Staubli VAL3: userPage.pjx

--- userPage.pjx ---
Parameters version=s7.6.3 stackSize=5000 millimeterUnit=true
Program file=changeTrsf.pgx
Program file=changeValue.pgx
Program file=clear.pgx
Program file=divideString.pgx
Program file=editNumField.pgx
Program file=findPos.pgx
Program file=getListPosition.pgx
Program file=getMenu.pgx
Program file=getView.pgx
Program file=insertDialog.pgx
Program file=insertDialog1.pgx
Program file=isListEmpty.pgx
Program file=leftPos.pgx
Program file=listadd.pgx
Program file=listcreate.pgx
Program file=listcursor.pgx
Program file=listdel.pgx
Program file=listempty.pgx
Program file=listevent.pgx
Program file=listframe.pgx
Program file=listins.pgx
Program file=listredraw.pgx
Program file=listupdate.pgx
Program file=listupdate1.pgx
Program file=midPos.pgx
Program file=nullKey.pgx
Program file=numCopy.pgx
Program file=printScroll.pgx
Program file=questionDialog.pgx
Program file=read.pgx
Program file=rightPos.pgx
Program file=scroll.pgx
Program file=selectNewField.pgx
Program file=setCenter.pgx
Program file=setMenu.pgx
Program file=setSizeList.pgx
Program file=setView.pgx
Program file=showBoolStatus.pgx
Program file=strfill.pgx
Program file=strfillchr.pgx
Program file=stringCopy.pgx
Program file=stringToArray.pgx
Program file=stringToFxArray.pgx
Program file=strlength.pgx
Program file=timerDialog.pgx
Program file=type.pgx
Program file=typeCenter.pgx
Program file=typeLen.pgx
Program file=typeMenu.pgx
Program file=yes_no.pgx
Program file=yes_no_cancel.pgx
Data file=userPage.dtx

--- changeTrsf.pgx ---
public program changeTrsf(trsf& x_tTrsf[], string x_sTitle, string x_sComment)
  local string l_sEvent
  local num l_nIndex
  local num l_nView
  local bool l_bRefresh
  local string l_sMessage
  local trsf l_tTrsf
  local string l_sItem
  local string l_sEmpty
  local point l_pPoint
  local tool l_tTool
  local num l_nAddon
  local num l_nDistanceX
  local num l_nDistanceY
  local bool l_bCheck
  local joint l_jPoint
begin
  logMsg("[KERNEL] INTERFACE:PAGE changeTrsf "+x_sTitle)
  // INIT all
  l_bRefresh=false
  l_nIndex=0
  l_nView=0
  call setSizeList(19,0,19,8)
  call setView(false)
  l_tTrsf=x_tTrsf
  //release the button
  call nullKey(nKey)
  // set the frame
  do
    cls()
    call type(0,12,x_sComment)
    call typeMenu(8,"OK")
    call listcreate(x_sTitle)
    l_sItem=("coord  X > "+toString(".2",l_tTrsf.x))
    call listadd(l_sItem)
    l_sItem=("coord  Y > "+toString(".2",l_tTrsf.y))
    call listadd(l_sItem)
    l_sItem=("coord  Z > "+toString(".2",l_tTrsf.z))
    call listadd(l_sItem)
    l_sItem=("coord RX > "+toString(".2",l_tTrsf.rx))
    call listadd(l_sItem)
    l_sItem=("coord RY > "+toString(".2",l_tTrsf.ry))
    call listadd(l_sItem)
    l_sItem=("coord RZ > "+toString(".2",l_tTrsf.rz))
    call listadd(l_sItem)
    // show the list
    nView=l_nIndex
    call listupdate(l_nIndex-l_nView)
    do
      l_nView=nView
      nKey=get()
      l_pPoint.trsf=l_tTrsf
      call listevent(nKey,l_nIndex,l_sEvent)
      switch nKey
        case 270
          //
          // clean the line
          call listcursor(nView,false)
          l_sEmpty=""
          switch l_nIndex
            case 0
              //  x-value
              call changeValue(l_tTrsf.x,0,0,10+40-nBottomX,nView+1,l_sEmpty)
            break
            case 1
              //  y-value
              call changeValue(l_tTrsf.y,0,0,10+40-nBottomX,nView+1,l_sEmpty)
            break
            case 2
              //  z-value
              call changeValue(l_tTrsf.z,0,0,10+40-nBottomX,nView+1,l_sEmpty)
            break
            case 3
              //  rx-value
              call changeValue(l_tTrsf.rx,0,0,10+40-nBottomX,nView+1,l_sEmpty)
            break
            case 4
              //  ry-value
              call changeValue(l_tTrsf.ry,0,0,10+40-nBottomX,nView+1,l_sEmpty)
            break
            case 5
              //  rz-value
              call changeValue(l_tTrsf.rz,0,0,10+40-nBottomX,nView+1,l_sEmpty)
            break
            case 6
              // addon
              l_nIndex=find(l_sEvent,">")
              call changeValue(l_nAddon,0,0,l_nIndex+1+2+nTopX,nView+nTopY+1,l_sEmpty)
            break
          endSwitch
          l_bRefresh=true
        break
        case 278
          // VALIDATE
          x_tTrsf=l_tTrsf
        break
      endSwitch
    until l_bRefresh==true or nKey==255 or nKey==278
    l_bRefresh=false
  until nKey==255 or nKey==278
  // check the key
  if nKey==278
    // validate
    x_tTrsf=l_tTrsf
  endIf
  // release the resource
  call nullKey(nKey)
end

--- changeValue.pgx ---
public program changeValue(num& x_nValue[], num x_nMin, num x_nMax, num x_nX, num x_nY, string& x_sItems[])
  local num l_nOldValue[2]
  local string l_sItem
  local string l_sMessage
  local bool l_bComma
  local string l_sEmpty
begin
  //---------------------------------
  // Staubli copyright 2005
  //                By toneage
  //[Public]-------------------------
  //
  // x_nValue:  num to change
  // x_nMax:    max value
  // x_nMin:    min value
  // x_nX:      X position
  // x_nY:      Y position
  // x_sItems   message
  //
  // look if the value is between max and min
  //
  if x_nMin>x_nMax
    return
  endIf
  //
  // print the line in white
  //
  // call listCleanLine()
  //
  call nullKey(nKey)
  l_nOldValue[1]=round(x_nValue)
  x_nValue=(round(x_nValue*100))/100
  l_nOldValue=x_nValue
  // check if is using the comma or not
  if l_nOldValue!=l_nOldValue[1]
    l_bComma=true
  else
    l_bComma=false
  endIf
  // start
  call clear(0,13)
  do
    if x_sItems==""
      //
      //  use the get num
      //
      if l_bComma
        call strfill(l_sEmpty,len(toString(".2",x_nValue)),l_sEmpty)
      else
        call strfill(l_sEmpty,len(toString("",x_nValue)),l_sEmpty)
      endIf
      call type(x_nX,x_nY,l_sEmpty)
      gotoxy(x_nX,x_nY)
      nKey=get(x_nValue)
      // check the comma again
      if round(x_nValue)!=x_nValue
        l_bComma=true
      endIf
      //
      // CHECK for MIN MAX VALUE
      //
      if x_nMax!=x_nMin or x_nMin!=0
        if x_nValue>x_nMax
          //
          // ask if you want to continue
          //
          popUpMsg("MAX: "+toString(".2",x_nMax))
          x_nValue=l_nOldValue
          //x_nValue=x_nMax
          nKey=-1
        else
          if x_nValue<x_nMin
            //
            popUpMsg("MIN: "+toString(".2",x_nMin))
            //x_nValue=x_nMin
            x_nValue=l_nOldValue
            nKey=-1
          endIf
        endIf
      endIf
      //
      // UPDATE THE VALUE
      //
      if l_bComma
        call type(x_nX,x_nY,toString(".2",x_nValue))
      else
        call type(x_nX,x_nY,toString("",x_nValue))
      endIf
    else
      //
      // STRING CHOICE
      //
      // show a list if there is the place
      call setSizeList(x_nX-1,max(0,x_nY-1),40-x_nX-1,min(13-x_nY,size(x_sItems)))
      call listcreate("")
      call listadd(x_sItems)
      call selectNewField(x_nValue,x_nValue,0)
      do
        nKey=get()
        call listevent(nKey,x_nValue,l_sItem)
      until nKey==270 or nKey==255
    endIf
  until nKey==270 or nKey==255
  if nKey==255
    bUseEscape=true
    x_nValue=l_nOldValue
    if x_sItems!=""
      x_sItems=x_sItems[l_nOldValue]
    endIf
  else
    bUseEscape=false
  endIf
end

--- insertDialog1.pgx ---
public program insertDialog1(string x_sMsg, num& x_nItem[], num x_nMin, num x_nMax)
  local num l_nStartLine
  local num l_nLine
  local num i
  local num l_nPX
  local num l_nPY
  local string l_sItem
  local string l_sMessage
  local string l_sEmpty
begin
  //
  // modify the x_sItem, using a min max range
  //
  if watch(bShowDialog==false,3)==false
    bShowDialog=false
    return
  else
    setMutex(bShowDialog)
    // clear the line
    call clear(0,13)
    // look for the comma
    if round(x_nItem)!=x_nItem
      l_sItem=toString(".2",x_nItem)
    else
      l_sItem=toString("",x_nItem)
    endIf
    // print the line
    l_sItem=x_sMsg+">"+l_sItem
    call stringCopy(l_sItem,sMessage)
    // divide the sentence
    call divideString(sMessage,l_nLine)
    l_nStartLine=round(5-l_nLine/2)
    // Start LINE
    call type(0,l_nStartLine-2,"┌──────────────────────────────────────┐")
    call type(0,l_nStartLine-1,"│                                      │")
    // write the message
    for i=0 to l_nLine
      //call type(,"                                      ")
      l_sMessage=sMessage[i]
      call typeCenter(i+l_nStartLine,l_sMessage,38,false)
      call type(0,l_nStartLine+i,"│"+l_sMessage+"│")
    endFor
    // end LINE
    call type(0,l_nStartLine+l_nLine+1,"│                                      │")
    call type(0,l_nStartLine+l_nLine+2,"└──────────────────────────────────────┘")
    l_nPX=find(l_sMessage,">")+2
    l_nPY=l_nStartLine+l_nLine
    // change the value
    call changeValue(x_nItem,x_nMin,x_nMax,l_nPX,l_nPY,l_sEmpty)
    //
    bShowDialog=false
    bUseRefresh=true
    //
  endIf
end

--- listcursor.pgx ---
public program listcursor(num pView (dimensions=1), bool pShow (dimensions=1))
  local num lX
  local num lY
  local string message
  local bool l_bEmpty
begin
  //
  // toneage Staubli Copyright 2005
  //
  call isListEmpty(l_bEmpty)
  if !l_bEmpty
    nView=pView
    lX=nTopX+1
    lY=nTopY+1+pView
    if (nView+nFirst)>(size(sItems)-1)
      call strfill(sItems[size(sItems)-1],nBottomX,message)
    else
      call strfill(sItems[max(0,nView+nFirst)],nBottomX,message)
    endIf
    gotoxy(lX,lY)
    if (pShow==true)
      setTextMode(1)
      put(message)
      setTextMode(0)
    else
      setTextMode(0)
      put(message)
    endIf
  endIf
end

--- listframe.pgx ---
program listframe(string pTitle (dimensions=1), num pX (dimensions=1), num pY (dimensions=1), num pDx (dimensions=1), num pDy (dimensions=1))
  local num lDx
  local num lDy
  local num lI
  local num lJ
  local string lStr
  local string lStrLine
  local num lValue
begin
  //
  // Staubli Copyright 2003 06 20
  //
  lStrLine="─────────────────────────────────────────"
  lDx=pDx
  lDy=pDy
  //Top
  lStr="┌"+mid(lStrLine,lDx,0)+"┐"
  gotoxy(pX,pY)
  put(lStr)
  lValue=pX+2
  //Title
  if pTitle!=""
    call leftPos("┤"+pTitle+"│",lDx+1,pTitle)
    gotoxy(pX+lDx-getDisplayLen(pTitle)+2,pY)
    put(pTitle)
  endIf
  //Containt
  for lJ=1 to lDy
    lValue=pY+lJ
    lStr="│"
    gotoxy(pX,lValue)
    put(lStr)
    gotoxy(pX+lDx+1,lValue)
    put(lStr)
  endFor
  //Bottom
  lValue=pY+lJ
  lStr="└"+mid(lStrLine,lDx,0)+"┘"
  gotoxy(pX,lValue)
  put(lStr)
end

--- listupdate1.pgx ---
public program listupdate1(num pFirst)
  local num lI
  local num lLen
  local string lStr
  local string lStr2
  local num lValue
  local num lView
  local num lX
  local num lY
  local num l_nSize
  local bool l_bEmpty
begin
  //
  // insert into the box all the data
  //
  // to prevent a negative value
  if pFirst>0
    nFirst=pFirst
  else
    nFirst=0
  endIf
  // save the coordinate
  lValue=nBottomY-1
  // check the overFlow
  l_nSize=size(sItems)-1
  if (nFirst+nView>l_nSize)
    // reset the value
    nFirst=nView=0
  endIf
  lI=0
  // check the unKnow poblem
  if l_nSize<lValue
    if nFirst!=0
      nView=nView+nFirst
      nFirst=0
    endIf
  endIf
  do
    lX=nTopX+1
    lY=nBottomY+lI-1
    lY=nTopY+lI+1
    lLen=nBottomX
    if ((lI+nFirst)<size(sItems))
      // print the item
      if (l_nSize>=0)
        lStr=mid(sItems[(lI+nFirst)],lLen,0)
      endIf
    else
      // print the blank line
      lStr="                                        "
    endIf
    // fill the line
    call strfill(lStr,lLen,lStr2)
    gotoxy(lX,lY)
    put(lStr2)
    lI=lI+1
  until (lI>lValue)
  // underlien the actual line
  call isListEmpty(l_bEmpty)
  if !l_bEmpty
    call listcursor(nView,false)
  else
    call listcursor(nView,false)
    nView=0
    nFirst=0
  endIf
  // print the scroll
  call printScroll()
end

--- numCopy.pgx ---
public program numCopy(num& x_nCopy[] (dimensions=1), num& x_nPaste[] (dimensions=1))
// Copy all the value from the x_nCopy to x_nPaste
  local num i
  local num l_nSize
begin
  // Copy all the value from the first element to the second one
  //
  // redim the Paste String ARRAY
  //
  if size(x_nPaste)!=size(x_nCopy)
    resize(x_nPaste,1,size(x_nCopy))
  endIf
  // COPY ALL THE FIELD
  for i=0 to (size(x_nCopy)-1)
    x_nPaste[i]=x_nCopy[i]
  endFor
end

--- printScroll.pgx ---
program printScroll()
  local num i
  local num lX
  local num lY
begin
  //
  // put the scroll
  //
  //if size(sItems)>nBottomY
  // find the percentage
  //windows style
  //i=(size(sItems)-nBottomY+1)/(nFirst+1)
  // nokia style
  i=(size(sItems))/(nFirst+nView+1)
  lX=nTopX+nBottomX+1
  lY=roundUp((nBottomY)/i+nTopY)
  for i=nTopY+1 to nBottomY
    gotoxy(lX,i)
    if (i==nTopY+1 and nFirst!=0)or(i==nBottomY and nFirst<=size(sItems)-1-(nBottomY-nTopY))and size(sItems)>nBottomY
      // show more items
      put("+")
    else
      put("│")
    endIf
  endFor
  //endIf
end

--- scroll.pgx ---
public program scroll(num x_nX (dimensions=1), num x_nY (dimensions=1), num x_nDim (dimensions=1), num x_nPos (dimensions=1))
// create a scroll bar
  local string l_sMessage
  local string l_sLine
  local num l_nPos
  local string l_sScrool
begin
  // use the scroll
  if x_nPos>0 and x_nPos<=100
    l_nPos=round(x_nDim*x_nPos/100)
    if l_nPos>0
      // make the scroll
      call strfill(l_sScrool,l_nPos,l_sScrool)
      call strfillchr(l_sScrool,l_sScrool,"■")
    endIf
    // make the line
    call strfill(l_sLine,x_nDim-l_nPos,l_sLine)
    call strfillchr(l_sLine,l_sLine,"─")
    l_sMessage="└"+l_sScrool+l_sLine+"┘"
    // show the line
    call type(x_nX,x_nY,l_sMessage)
  endIf
end

--- setMenu.pgx ---
public program setMenu(string& x_sMenuName[] (dimensions=1), bool x_bShowName (dimensions=1), num x_nY (dimensions=1))
// Show the
  local num i
begin
  //
  // usage
  // menuname"choice1,choise2,..choise7,choice8"
  //
  // the page will start from the y- line
  //
  //
  if size(x_sMenuName)<10
    for i=0 to (size(x_sMenuName)-1)
      if x_sMenuName[i]!="" and x_sMenuName[i]!=" "
        if x_bShowName==false
          call typeMenu(i+1,"F"+toString("1",i+1))
        else
          call typeMenu(i+1,x_sMenuName[i])
        endIf
        if x_nY!=-1
          call type(0,i+x_nY,("F"+(toString("1",i+1)+" "+x_sMenuName[i])))
        endIf
      endIf
    endFor
  endIf
end

--- stringCopy.pgx ---
public program stringCopy(string& x_sCopy[] (dimensions=1), string& x_sPaste[] (dimensions=1))
// Copy all the value from the x_sCopy to x_sPaste
  local num i
  local num l_nSize
begin
  // Copy all the value from the first element to the second one
  //
  // redim the Paste String ARRAY
  //
  //l_nSize=size(x_sPaste)
  if size(x_sPaste)!=size(x_sCopy)
    resize(x_sPaste,1,size(x_sCopy))
  endIf
  //  if size(x_sCopy)>size(x_sPaste)
  //    for i=l_nSize to (size(x_sCopy)-1)
  //      insert(x_sPaste[i])
  //    endFor
  //  else
  //    if size(x_sCopy)<size(x_sPaste)
  //      for i=size(x_sCopy) to l_nSize-1
  //        delete(x_sPaste[size(x_sCopy)])
  //      endFor
  //    endIf
  //  endIf
  // COPY ALL THE FIELD
  for i=0 to (size(x_sCopy)-1)
    x_sPaste[i]=x_sCopy[i]
  endFor
end

--- stringToFxArray.pgx ---
public program stringToFxArray(string x_sString (dimensions=1), string& x_sArray[] (dimensions=1))
// copy one String into an ARRAY of String
  local num i
  local num l_nItem
  local string l_sChar
  local string l_sEmpty
begin
  // define the char use to divide the items
  // PRIORITY
  //  ^
  //  ;
  //  ,
  //
  if find(x_sString,"^")==-1
    if find(x_sString,";")==-1
      l_sChar=","
    else
      l_sChar=";"
    endIf
  else
    l_sChar="^"
  endIf
  // init the X_sArray
  l_nItem=0
  do
    i=find(x_sString,l_sChar)
    // look if was found
    if i!=-1
      // PUT INSIDE THE ARRAY THE STRING
      x_sArray[l_nItem]=left(x_sString,i)
      x_sString=delete(x_sString,i+1,0)
    else
      // look if is empty or not
      if len(x_sString)>0
        x_sArray[l_nItem]=(x_sString)
      else
        x_sArray[l_nItem]=""
      endIf
    endIf
    l_nItem=l_nItem+1
  until i==-1
  // fill with empty field for the rest
  for i=l_nItem to size(x_sArray)-1 step 1
    x_sArray[i]=""
  endFor
end

--- timerDialog.pgx ---
public program timerDialog(string x_sMsg, num x_nTime)
  local num l_nTime
  local num l_nStartLine
  local num l_nLine
  local num i
  local string l_sMessage
begin
  //
  // use for other task
  //
  if watch(bShowDialog==false,3)==false
    bShowDialog=false
    return
  else
    setMutex(bShowDialog)
    //
    //call listempty()
    //
    l_nTime=clock()
    call stringCopy(x_sMsg,sMessage)
    call divideString(sMessage,l_nLine)
    l_nStartLine=round(5-l_nLine/2)
    do
      // Start LINE
      call type(0,l_nStartLine-2,"┌──────────────────────────────────────┐")
      call type(0,l_nStartLine-1,"│                                      │")
      // write the message
      for i=0 to l_nLine
        call type(0,l_nStartLine+i,"")
        call type(39,l_nStartLine+i,"")
        //call typeCenter(i+l_nStartLine,sMessage[i],38,false)
        l_sMessage=sMessage[i]
        call typeCenter(i+l_nStartLine,l_sMessage,38,false)
        call type(0,l_nStartLine+i,"│"+l_sMessage+"│")
      endFor
      // end LINE
      call type(0,l_nStartLine+l_nLine+1,"│                                      │")
      call type(0,l_nStartLine+l_nLine+2,"└──────────────────────────────────────┘")
      // release
      if x_nTime==0
        delay(0.1)
      else
        delay(0)
      endIf
    until (clock()-l_nTime)>=x_nTime
    //
    bShowDialog=false
    bUseRefresh=true
  endIf
end
